///FUNCTION_BLOCK PUBLIC FB_IBuffer IMPLEMENTS IBuffer
FUNCTION_BLOCK FB_IBuffer EXTENDS FB_CtrlBase IMPLEMENTS IBuffer

// This is a Dummy-FB, used for the interface (IBuffer) to the buffer-modules

PROPERTY MaxCapacity : DINT
GET
END_GET
END_PROPERTY

PROPERTY NumOfHangers : DINT
GET
END_GET
END_PROPERTY

END_FUNCTION_BLOCK

(* stored: Version 1.1.0.1, ProductVersion 3.1.0.19
   POU FB_IBuffer: Id {ac812cbe-1f8b-47d1-861d-77e5638b9fdc}
   Property MaxCapacity: Id {b708dd4b-5b49-4fd6-ab56-49c1ad8d751e}
   Get Get: Id {7a16a80c-12db-4e9b-a2d5-d16684b8459d}
   Property NumOfHangers: Id {64648448-e502-41cf-bc7b-35ef7e411c3a}
   Get Get: Id {82d4a0d6-e187-412c-801d-93bbbab40c16} *)
